ABB RobotStudio station: Assignment2_task#4.rspag

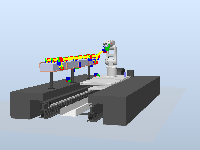
--- station ---
Station Assignment2_task#4 (saved by RobotStudio 20.1.9014.1)
Controller Controller5, task T_ROB1: task frame (RAPID world) sits at (0, 270, 397.5) mm, rotated rx 0 ry 0 rz 180 deg in the station
Controller Controller5
  mechanical unit ROB_1: IRB120_3_58__01, 6 joints, base frame (0, 0, 0) mm
  mechanical unit TRACK: RTT_Bobin_1_7, 1 joints, base frame (0, 0, 0) mm
Layout (positions relative to the parent item):
  - RTT_Bobin_1_7 [mechanism] at (0, 270, 0) mm, rotated rx 0 ry 0 rz 180 deg; joint values [0] (rad or m)
      links: Base, Link1
  - IRB120_3_58__01 [mechanism, from Robots\IRB120_3_58_G_01.rslib] at (0, 270, 397.5) mm, rotated rx 0 ry 0 rz 180 deg; joint values [0, 0, 0, 0, 0.5236, 0] (rad or m)
  - AssemblyDrillbit [part] at (-362.14, 195.92, 1033.34) mm, rotated rx -90 ry 60 rz 0 deg
  - Task4_Part [part] at (-2000, 570, 647.5) mm, rotated rx 90 ry 0 rz 0 deg
  - FloorTop [part] at (700, 0, 0) mm
  - FloorBase [part]
  - FloorBase_2 [part] at (-1600, 540, 0) mm, rotated rx 0 ry 0 rz 180 deg
  - FloorTop_2 [part] at (-2300, 540, 0) mm, rotated rx 0 ry 0 rz 180 deg
  - BaseSupport [part]
  - BackSupport [part]
  - LegSupport1 [part]
  - LegBase1 [part]
  - LegSupport2 [part] at (-850, 0, 0) mm
  - LegBase2 [part] at (-850, 0, 0) mm
  - LegBase3 [part] at (850, 0, 0) mm
  - LegSupport3 [part] at (850, 0, 0) mm
  - MaterialBackSupport1 [part]
  - SideSupport1 [part]
  - SideSupport2 [part] at (-500, 0, 0) mm
  - SideSupport3 [part] at (500, 0, 0) mm
  - EndSupport [part]
Attachment: IRB120_3_58__01 is attached to RTT_Bobin_1_7 / Link1
Attachment: AssemblyDrillbit is attached to IRB120_3_58__01 / Link6
Attachment: FloorTop is attached to FloorBase
Attachment: FloorTop_2 is attached to FloorBase_2
Attachment: BackSupport is attached to BaseSupport
Attachment: LegSupport1 is attached to LegBase1
Attachment: LegBase2 is attached to LegSupport2
Attachment: LegBase3 is attached to LegSupport3
Attachment: BaseSupport is attached to LegSupport1
Attachment: SideSupport1 is attached to BaseSupport
Attachment: EndSupport is attached to MaterialBackSupport1

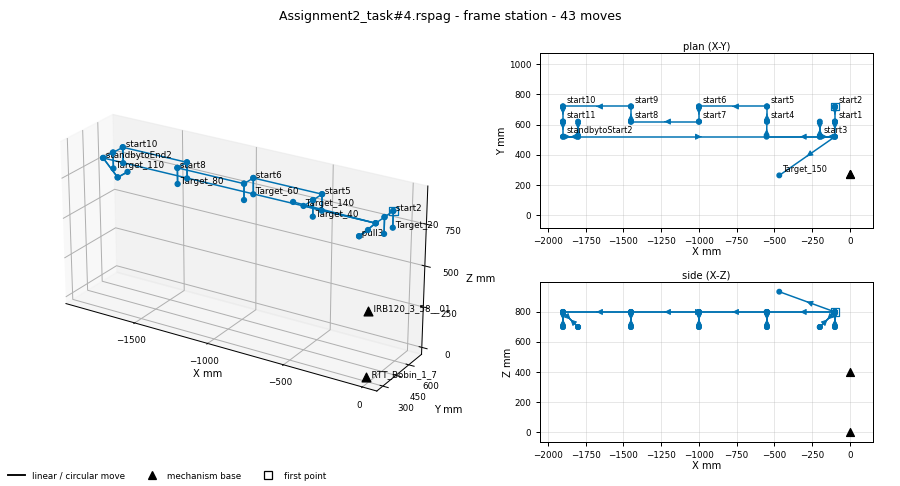
[picture p0: tool path of Assignment2_task#4.rspag in frame station, 43 of 43 moves have a stored position in this frame; points joined in program order, loops and branches not executed]
--- Backups/Controller5/RAPID/TASK1/PROGMOD/CalibData.mod ---
MODULE CalibData
    TASK PERS tooldata Drill:=[TRUE,[[0,6,120],[1,0,0,0]],[1,[0,0,1],[1,0,0,0],0,0,0]];
    TASK PERS wobjdata Task4:=[FALSE,TRUE,"",[[0,-300,0],[1,0,0,0]],[[0,0,0],[1,0,0,0]]];
    TASK PERS wobjdata Workobject_1:=[FALSE,TRUE,"",[[-700,-570,-130],[0,1,0,0]],[[0,0,0],[1,0,0,0]]];
    TASK PERS wobjdata Workobject_2:=[FALSE,TRUE,"",[[800,-570,-30],[1,0,0,0]],[[0,0,0],[1,0,0,0]]];
    TASK PERS wobjdata ObjectSupport:=[FALSE,TRUE,"",[[0,-400,250],[0,1,0,0]],[[0,0,0],[1,0,0,0]]];
    TASK PERS wobjdata objectSupport2:=[FALSE,TRUE,"",[[0,-515,250],[1,0,0,0]],[[0,0,0],[1,0,0,0]]];
    TASK PERS wobjdata LegSupport:=[FALSE,TRUE,"",[[1000,-400,235],[0,1,0,0]],[[0,0,0],[1,0,0,0]]];
    TASK PERS wobjdata MaterialSupporter:=[FALSE,TRUE,"",[[1000,-285,250],[0,0,0,1]],[[0,0,0],[1,0,0,0]]];
    TASK PERS wobjdata MaterialSupporter2:=[FALSE,TRUE,"",[[-15,-400,250],[1,0,0,0]],[[0,0,0],[1,0,0,0]]];
ENDMODULE

--- Backups/Controller5/RAPID/TASK1/PROGMOD/Module1.mod ---
MODULE Module1
        CONST robtarget Target_130:=[[100.000011963,-250.000018925,399.999968915],[0.000000014,0.707106776,0.707106787,0.000000006],[-1,0,0,0],[0,9E+09,9E+09,9E+09,9E+09,9E+09]];
    CONST robtarget start1:=[[100,-50,400],[0,0.707106781,0.707106781,0],[-1,0,0,0],[0,9E+09,9E+09,9E+09,9E+09,9E+09]];
    CONST robtarget Target_10:=[[100,-50,300],[0,0.707106781,0.707106781,0],[-1,0,0,0],[0,9E+09,9E+09,9E+09,9E+09,9E+09]];
    CONST robtarget lift1:=[[100,-50,400],[0,0.707106781,0.707106781,0],[-1,0,0,0],[0,9E+09,9E+09,9E+09,9E+09,9E+09]];
    CONST robtarget start2:=[[100,-150,400],[0,0.707106781,0.707106781,0],[-1,0,0,0],[0,9E+09,9E+09,9E+09,9E+09,9E+09]];
    CONST robtarget Target_20:=[[100,-150,300],[0,0.707106781,0.707106781,0],[-1,0,0,0],[0,9E+09,9E+09,9E+09,9E+09,9E+09]];
    CONST robtarget lift2:=[[100,-150,400],[0,0.707106781,0.707106781,0],[-1,0,0,0],[0,9E+09,9E+09,9E+09,9E+09,9E+09]];
    CONST robtarget standbyToStart1:=[[100,50,400],[0,0.707106781,0.707106781,0],[-1,0,0,0],[0,9E+09,9E+09,9E+09,9E+09,9E+09]];
    CONST robtarget start3:=[[200,50,300],[0.5,0.5,0.5,-0.5],[-1,-2,1,0],[0,9E+09,9E+09,9E+09,9E+09,9E+09]];
    CONST robtarget Target_30:=[[200,-50,300],[0.5,0.5,0.5,-0.5],[-1,-2,1,0],[0,9E+09,9E+09,9E+09,9E+09,9E+09]];
    CONST robtarget pull3:=[[200,50,300],[0.5,0.5,0.5,-0.5],[-1,-2,1,0],[0,9E+09,9E+09,9E+09,9E+09,9E+09]];
    CONST robtarget standbyToEnd1:=[[100,50,400],[0,0.707106781,0.707106781,0],[-1,0,0,0],[0,9E+09,9E+09,9E+09,9E+09,9E+09]];
    CONST robtarget Target_140:=[[552.545588746,-250.000018925,399.999968915],[0.000000014,0.707106776,0.707106787,0.000000006],[-1,0,0,0],[418.88,9E+09,9E+09,9E+09,9E+09,9E+09]];
    CONST robtarget start4:=[[550,-50,400],[0,0.707106781,0.707106781,0],[-1,0,0,0],[418.88,9E+09,9E+09,9E+09,9E+09,9E+09]];
    CONST robtarget Target_40:=[[550,-50,300],[0,0.707106781,0.707106781,0],[-1,0,0,0],[418.88,9E+09,9E+09,9E+09,9E+09,9E+09]];
    CONST robtarget lift4:=[[550,-50,400],[0,0.707106781,0.707106781,0],[-1,0,0,0],[418.88,9E+09,9E+09,9E+09,9E+09,9E+09]];
    CONST robtarget start5:=[[550,-150,400],[0,0.707106781,0.707106781,0],[-1,0,0,0],[418.88,9E+09,9E+09,9E+09,9E+09,9E+09]];
    CONST robtarget Target_50:=[[550,-150,300],[0,0.707106781,0.707106781,0],[-1,0,0,0],[418.88,9E+09,9E+09,9E+09,9E+09,9E+09]];
    CONST robtarget lift5:=[[550,-150,400],[0,0.707106781,0.707106781,0],[-1,0,0,0],[418.88,9E+09,9E+09,9E+09,9E+09,9E+09]];
    CONST robtarget start6:=[[1000,-150,400],[0,0.707106781,0.707106781,0],[-1,0,0,0],[802.85,9E+09,9E+09,9E+09,9E+09,9E+09]];
    CONST robtarget Target_60:=[[1000,-150,300],[0,0.707106781,0.707106781,0],[-1,0,0,0],[802.85,9E+09,9E+09,9E+09,9E+09,9E+09]];
    CONST robtarget lift6:=[[1000,-150,400],[0,0.707106781,0.707106781,0],[-1,0,0,0],[802.85,9E+09,9E+09,9E+09,9E+09,9E+09]];
    CONST robtarget start7:=[[1000,-50,400],[0,0.707106781,0.707106781,0],[-1,0,0,0],[802.85,9E+09,9E+09,9E+09,9E+09,9E+09]];
    CONST robtarget Target_70:=[[1000,-50,300],[0,0.707106781,0.707106781,0],[-1,0,0,0],[802.85,9E+09,9E+09,9E+09,9E+09,9E+09]];
    CONST robtarget lift7:=[[1000,-50,400],[0,0.707106781,0.707106781,0],[-1,0,0,0],[802.85,9E+09,9E+09,9E+09,9E+09,9E+09]];
    CONST robtarget start8:=[[1450,-50,400],[0,0.707106781,0.707106781,0],[-1,0,0,0],[1309,9E+09,9E+09,9E+09,9E+09,9E+09]];
    CONST robtarget Target_80:=[[1450,-50,300],[0,0.707106781,0.707106781,0],[-1,0,0,0],[1309,9E+09,9E+09,9E+09,9E+09,9E+09]];
    CONST robtarget lift8:=[[1450,-50,400],[0,0.707106781,0.707106781,0],[-1,0,0,0],[1309,9E+09,9E+09,9E+09,9E+09,9E+09]];
    CONST robtarget start9:=[[1450,-150,400],[0,0.707106781,0.707106781,0],[-1,0,0,0],[1309,9E+09,9E+09,9E+09,9E+09,9E+09]];
    CONST robtarget Target_90:=[[1450,-150,300],[0,0.707106781,0.707106781,0],[-1,0,0,0],[1309,9E+09,9E+09,9E+09,9E+09,9E+09]];
    CONST robtarget lift9:=[[1450,-150,400],[0,0.707106781,0.707106781,0],[-1,0,0,0],[1309,9E+09,9E+09,9E+09,9E+09,9E+09]];
    CONST robtarget start10:=[[1900,-150,400],[0,0.707106781,0.707106781,0],[-1,0,0,0],[1692.97,9E+09,9E+09,9E+09,9E+09,9E+09]];
    CONST robtarget Target_100:=[[1900,-150,300],[0,0.707106781,0.707106781,0],[-1,0,0,0],[1692.97,9E+09,9E+09,9E+09,9E+09,9E+09]];
    CONST robtarget lift10:=[[1900,-150,400],[0,0.707106781,0.707106781,0],[-1,0,0,0],[1692.97,9E+09,9E+09,9E+09,9E+09,9E+09]];
    CONST robtarget start11:=[[1900,-50,400],[0,0.707106781,0.707106781,0],[-1,0,0,0],[1692.97,9E+09,9E+09,9E+09,9E+09,9E+09]];
    CONST robtarget Target_110:=[[1900,-50,300],[0,0.707106781,0.707106781,0],[-1,0,0,0],[1692.97,9E+09,9E+09,9E+09,9E+09,9E+09]];
    CONST robtarget lift11:=[[1900,-50,400],[0,0.707106781,0.707106781,0],[-1,0,0,0],[1692.97,9E+09,9E+09,9E+09,9E+09,9E+09]];
    CONST robtarget standbytoStart2:=[[1900,50,400],[0,0.707106781,0.707106781,0],[-1,0,0,0],[1692.97,9E+09,9E+09,9E+09,9E+09,9E+09]];
    CONST robtarget start12:=[[1800,50,300],[0.5,0.5,0.5,-0.5],[-1,-2,1,0],[1518.44,9E+09,9E+09,9E+09,9E+09,9E+09]];
    CONST robtarget Target_120:=[[1800,-50,300],[0.5,0.5,0.5,-0.5],[-1,-2,1,0],[1692.97,9E+09,9E+09,9E+09,9E+09,9E+09]];
    CONST robtarget pull12:=[[1800,50,300],[0.5,0.5,0.5,-0.5],[-1,-2,1,0],[1518.44,9E+09,9E+09,9E+09,9E+09,9E+09]];
    CONST robtarget standbytoEnd2:=[[1900,50,400],[0,0.707106781,0.707106781,0],[-1,0,0,0],[1692.97,9E+09,9E+09,9E+09,9E+09,9E+09]];
    CONST robtarget Target_150:=[[-531.723130631,-406.000012107,-299.000005122],[0,0.500000001,0,0.866025403],[0,-1,0,0],[0,9E+09,9E+09,9E+09,9E+09,9E+09]];
!***********************************************************
    !
    ! Module:  Module1
    !
    ! Description:
    !   <Insert description here>
    !
    ! Author: adityaaaap
    !
    ! Version: 1.0
    !
    !***********************************************************


    !***********************************************************
    !
    ! Procedure main
    !
    !   This is the entry point of your program
    !
    !***********************************************************
    PROC main()
        !Add your code here
        Path_10;
    ENDPROC
    PROC Path_10()
        MoveL start2,v100,z10,Drill\WObj:=Task4;
        MoveL Target_20,v100,z10,Drill\WObj:=Task4;
        MoveL lift2,v100,z10,Drill\WObj:=Task4;
        MoveL start1,v100,z10,Drill\WObj:=Task4;
        MoveL Target_10,v100,z10,Drill\WObj:=Task4;
        MoveL lift1,v100,z10,Drill\WObj:=Task4;
        MoveL standbyToStart1,v100,z10,Drill\WObj:=Task4;
        MoveL start3,v100,z10,Drill\WObj:=Task4;
        MoveL Target_30,v100,z10,Drill\WObj:=Task4;
        MoveL pull3,v100,z10,Drill\WObj:=Task4;
        MoveL standbyToEnd1,v100,z10,Drill\WObj:=Task4;
        MoveL Target_140,v100,z10,Drill\WObj:=wobj0;
        MoveL start4,v100,z10,Drill\WObj:=Task4;
        MoveL Target_40,v100,z10,Drill\WObj:=Task4;
        MoveL lift4,v100,z10,Drill\WObj:=Task4;
        MoveL start5,v100,z10,Drill\WObj:=Task4;
        MoveL Target_50,v100,z10,Drill\WObj:=Task4;
        MoveL lift5,v100,z10,Drill\WObj:=Task4;
        MoveL start6,v100,z10,Drill\WObj:=Task4;
        MoveL Target_60,v100,z10,Drill\WObj:=Task4;
        MoveL lift6,v100,z10,Drill\WObj:=Task4;
        MoveL start7,v100,z10,Drill\WObj:=Task4;
        MoveL Target_70,v100,z10,Drill\WObj:=Task4;
        MoveL lift7,v100,z10,Drill\WObj:=Task4;
        MoveL start8,v100,z10,Drill\WObj:=Task4;
        MoveL Target_80,v100,z10,Drill\WObj:=Task4;
        MoveL lift8,v100,z10,Drill\WObj:=Task4;
        MoveL start9,v100,z10,Drill\WObj:=Task4;
        MoveL Target_90,v100,z10,Drill\WObj:=Task4;
        MoveL lift9,v100,z10,Drill\WObj:=Task4;
        MoveL start10,v100,z10,Drill\WObj:=Task4;
        MoveL Target_100,v100,z10,Drill\WObj:=Task4;
        MoveL lift10,v100,z10,Drill\WObj:=Task4;
        MoveL start11,v100,z10,Drill\WObj:=Task4;
        MoveL Target_110,v100,z10,Drill\WObj:=Task4;
        MoveL lift11,v100,z10,Drill\WObj:=Task4;
        MoveL standbytoStart2,v100,z10,Drill\WObj:=Task4;
        MoveL start12,v100,z10,Drill\WObj:=Task4;
        MoveL Target_120,v100,z10,Drill\WObj:=Task4;
        MoveL pull12,v100,z10,Drill\WObj:=Task4;
        MoveL standbytoEnd2,v100,z10,Drill\WObj:=Task4;
        MoveL Target_130,v100,z10,Drill\WObj:=wobj0;
        MoveL Target_150,v100,z10,Drill\WObj:=LegSupport;
    ENDPROC
ENDMODULE
